FUNCTION func_f2: BOOL
VAR_INPUT
    farg_f2_p: BOOL;
END_VAR


        func_f2 := ifExprFunc2(farg_f2_p:=farg_f2_p);
RETURN;

END_FUNCTION

(* stored: ProductVersion 3.1.0.18, Version 1.1.0.1 *)
